# EPICS substitutions: EUROTHRM/EUROTHRM-IOC-01App/Db/devEurothrmA07.substitutions
# Note: this file is generated by generate_substitutions.py
file devEurothrm.template {
pattern { P, GAD, LAD, MODBUS_PV, MODBUS_SP, MODBUS_P, MODBUS_I, MODBUS_D, MODBUS_HS, MODBUS_LS, MODBUS_AT, MODBUS_HO, MODBUS_OP }
{ "\$(P)", "0", "7", "6145", "6146", "6150", "6152", "6153", "6255", "6256", "6414", "6174", "6147" }
}
